// TIA Portal V19 export
DATA_BLOCK "GET_DB"   // DB7
// stored: InstanceOfName GET_SFB, OfSystemLibElement GET, OfSystemLibVersion 1.3
"GET_SFB"
   // VAR_INPUT
   //    REQ : Bool;
   //    ID : Word;
   // END_VAR
   // VAR_OUTPUT
   //    NDR : Bool;
   //    ERROR : Bool;
   //    STATUS : Word;
   // END_VAR
   // VAR_IN_OUT
   //    ADDR_1 : Remote;
   //    ADDR_2 : Remote;
   //    ADDR_3 : Remote;
   //    ADDR_4 : Remote;
   //    RD_1 : Variant;
   //    RD_2 : Variant;
   //    RD_3 : Variant;
   //    RD_4 : Variant;
   // END_VAR
BEGIN
END_DATA_BLOCK
